(* IEC 61131-3 sources: T4Exjobb/Sigma/Stations/MachineControl/MachineControl/Class/UserAlarmGenerator, 1 file *)

(* ---- UserAlarmGenerator.st ---- *)
(*!
<Class
	Name               = "UserAlarmGenerator"
	Revision           = "1.1"
	RealtimeTask       = "false"
	CyclicTask         = "true"
	BackgroundTask     = "false"
	Sigmatek           = "false"
	OSInterface        = "false"
	HighPriority       = "false"
	Automatic          = "false"
	UpdateMode         = "Prescan"
	SharedCommandTable = "true"
	Objectsize         = "(420,240)"
	Comment            = "Class checks status of a Server and initiates a write (to an alarm server) if necessary">
	<Channels>
		<Server Name="ClassSvr" Visualized="false" Initialize="false" WriteProtected="true" Retentive="false" Comment="class server"/>
		<Client Name="In_mode" Required="true" Internal="false" Comment="0= create alarm if  In_status is LOW&#13;&#10;1= create alarm if  In_status is HIGH"/>
		<Client Name="In_status" Required="true" Internal="false" Comment="status to be watched for alarming"/>
		<Client Name="Out_alarm" Required="true" Internal="false" Comment="1= ALARM (status is not OK)"/>
	</Channels>
	<Dependencies>
		<Files>
			<File Path=".\Class\UserAlarmGenerator\UserAlarmGenerator_de.pdf"/>
			<File Path=".\Class\UserAlarmGenerator\UserAlarmGenerator_en.pdf"/>
		</Files>
	</Dependencies>
	<RevDoku>
		<Owner Company="Sigmatek" Author="KaiAnd"/>
		<Dokumentation Revision="1.1" Date="2016-10-10" Author="HubChr" Company="Sigmatek" Description="Added documentation pdfs."/>
		<Dokumentation Revision="1.0" Date="2016-05-24" Author="KaiAnd" Company="Sigmatek" Description="Creation."/>
	</RevDoku>
</Class>
*)
UserAlarmGenerator : CLASS
  //Servers:
	ClassSvr 	: SvrChCmd_DINT;
  //Clients:
	Out_alarm 	: CltCh_DINT;
	In_status 	: CltCh_DINT;
	In_mode 	: CltCh_DINT;
  //Variables:
  //Functions:

	FUNCTION VIRTUAL GLOBAL CyWork
		VAR_INPUT
			EAX 	: UDINT;
		END_VAR
		VAR_OUTPUT
			state (EAX) 	: UDINT;
		END_VAR;
  //Tables:
	FUNCTION @STD
		VAR_OUTPUT
			ret_code	: CONFSTATES;
		END_VAR;
	FUNCTION GLOBAL TAB @CT_;
END_CLASS;

FUNCTION VIRTUAL GLOBAL UserAlarmGenerator::CyWork
	VAR_INPUT
		EAX 	: UDINT;
	END_VAR
	VAR_OUTPUT
		state (EAX) 	: UDINT;
	END_VAR
  VAR
  	myAlarm : DINT;   // internal alarm
  END_VAR

  //----- visualize the clients -----------------
  Out_alarm := Out_alarm.Read();
  In_status := In_status.Read();
  In_mode   := In_mode.Read();

  //----- building the internal alarm -----------
  myAlarm := 0;
  if (In_mode = In_status) then
    myAlarm := 1;
  end_if;

  //----- write the output ----------------------
  if (myAlarm <> Out_alarm.Read()) then
      Out_alarm.Write(myAlarm);
  end_if;

	state := READY;

END_FUNCTION
